// TIA Portal V17 export
// export: Created 2023-12-22T15:05:26.061098Z, ExportSetting WithDefaults, DisplayName Totally Integrated Automation Portal, DisplayVersion V17, DisplayName TIA Portal Openness, DisplayVersion V17, DisplayName TIA Portal Version Control Interface, DisplayVersion V17, DisplayName STEP 7 Professional, DisplayVersion V17, DisplayName STEP 7 Safety, DisplayVersion V17, DisplayName WinCC Advanced, DisplayVersion V17
FUNCTION_BLOCK "Lock"   // FB2, LAD
{ S7_Optimized_Access := 'TRUE' }
VERSION : 0.1
// stored: AutoNumber true, IsIECCheckEnabled false, IsRetainMemResEnabled false, MemoryReserve 100, SetENOAutomatically false, UDAEnableTagReadback false
BEGIN

REGION Network 1: Блокировка электролизера
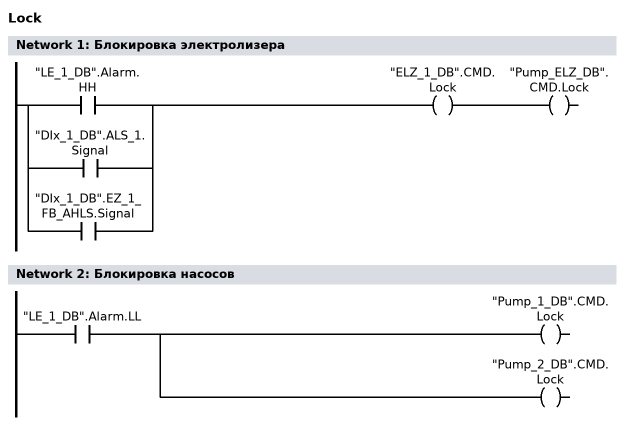
   RUNG wire#powerrail
      Contact( "LE_1_DB".Alarm.HH )
      wire#w1
      Coil( "ELZ_1_DB".CMD.Lock )
      Coil( "Pump_ELZ_DB".CMD.Lock )
   END_RUNG
   RUNG wire#powerrail
      Contact( "DIx_1_DB".ALS_1.Signal )
   END_RUNG wire#w1
   RUNG wire#powerrail
      Contact( "DIx_1_DB".EZ_1_FB_AHLS.Signal )
   END_RUNG wire#w1
   // the same network as SCL:
   "ELZ_1_DB".CMD.Lock := "LE_1_DB".Alarm.HH OR "DIx_1_DB".ALS_1.Signal OR "DIx_1_DB".EZ_1_FB_AHLS.Signal;
   "Pump_ELZ_DB".CMD.Lock := "ELZ_1_DB".CMD.Lock;
END_REGION

REGION Network 2: Блокировка насосов
   RUNG wire#powerrail
      Contact( "LE_1_DB".Alarm.LL )
      wire#w1
      Coil( "Pump_1_DB".CMD.Lock )
   END_RUNG
   RUNG wire#w1
      Coil( "Pump_2_DB".CMD.Lock )
   END_RUNG
   // the same network as SCL:
   "Pump_1_DB".CMD.Lock := "LE_1_DB".Alarm.LL;
   "Pump_2_DB".CMD.Lock := "LE_1_DB".Alarm.LL;
END_REGION
END_FUNCTION_BLOCK
